# EPICS substitutions: adsApp/Db/DUT_AxisStatus.substitutions
file "DUT_AxisStatus_v0_01.template"
{
pattern
{P,      PORT,      A, P, VP,     VI, VN }
{ADSTEST:,  ADS_1,  "", "", Main.M, 1,  stAxisStatus}
}
